FUNCTION_BLOCK LINE_MANAGER
  {SET_ATTRIBUTE(OpcUa, SERVICE)}
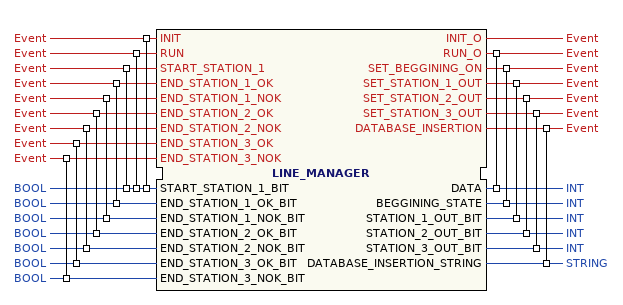
  EVENT_INPUT
    INIT WITH START_STATION_1_BIT;
    RUN WITH START_STATION_1_BIT;
    START_STATION_1 WITH START_STATION_1_BIT;
    END_STATION_1_OK WITH END_STATION_1_OK_BIT;
    END_STATION_1_NOK WITH END_STATION_1_NOK_BIT;
    END_STATION_2_OK WITH END_STATION_2_OK_BIT;
    END_STATION_2_NOK WITH END_STATION_2_NOK_BIT;
    END_STATION_3_OK WITH END_STATION_3_OK_BIT;
    END_STATION_3_NOK WITH END_STATION_3_NOK_BIT;
  END_EVENT
  EVENT_OUTPUT
    INIT_O;
    RUN_O WITH DATA;
    SET_BEGGINING_ON WITH BEGGINING_STATE;
    SET_STATION_1_OUT WITH STATION_1_OUT_BIT;
    SET_STATION_2_OUT WITH STATION_2_OUT_BIT;
    SET_STATION_3_OUT WITH STATION_3_OUT_BIT;
    DATABASE_INSERTION WITH DATABASE_INSERTION_STRING;
  END_EVENT
  VAR_INPUT
    START_STATION_1_BIT : BOOL; {SET_ATTRIBUTE(OpcUa, Variable.RUN)}
    END_STATION_1_OK_BIT : BOOL; {SET_ATTRIBUTE(OpcUa, Variable.RUN)}
    END_STATION_1_NOK_BIT : BOOL; {SET_ATTRIBUTE(OpcUa, Variable.RUN)}
    END_STATION_2_OK_BIT : BOOL; {SET_ATTRIBUTE(OpcUa, Variable.RUN)}
    END_STATION_2_NOK_BIT : BOOL; {SET_ATTRIBUTE(OpcUa, Variable.RUN)}
    END_STATION_3_OK_BIT : BOOL; {SET_ATTRIBUTE(OpcUa, Variable.RUN)}
    END_STATION_3_NOK_BIT : BOOL; {SET_ATTRIBUTE(OpcUa, Variable.RUN)}
  END_VAR
  VAR_OUTPUT
    DATA : INT; {SET_ATTRIBUTE(OpcUa, Variable.RUN)}
    BEGGINING_STATE : INT; {SET_ATTRIBUTE(OpcUa, Variable.RUN)}
    STATION_1_OUT_BIT : INT; {SET_ATTRIBUTE(OpcUa, Variable.RUN)}
    STATION_2_OUT_BIT : INT; {SET_ATTRIBUTE(OpcUa, Variable.RUN)}
    STATION_3_OUT_BIT : INT; {SET_ATTRIBUTE(OpcUa, Variable.RUN)}
    DATABASE_INSERTION_STRING : STRING; {SET_ATTRIBUTE(OpcUa, Variable.RUN)}
  END_VAR
END_FUNCTION_BLOCK
